{attribute 'c++_compatible'}
FUNCTION_BLOCK FB_ReadJSON IMPLEMENTS ITcJsonSaxHandler
VAR_INPUT
    myArrayInput1 : REFERENCE TO ARRAY[1..CONSt.STATION_NUMBER] OF DINT;
    myArrayInput2 : REFERENCE TO ARRAY[1..CONSt.STATION_NUMBER] OF DINT;
END_VAR
VAR_OUTPUT
END_VAR
VAR
    iArrayIndex : INT;
	iArrayNumber : INT := 0;
END_VAR

{attribute 'TcTypeSystem'}
{attribute 'no-analysis'}
{attribute 'c++_compatible'}
{attribute 'minimal_input_size' := '4'}
{attribute 'pack_mode' := '4'}
METHOD OnBool : HRESULT
VAR_INPUT
	value	: BOOL;
END_VAR
END_METHOD

{attribute 'TcTypeSystem'}
{attribute 'no-analysis'}
{attribute 'c++_compatible'}
{attribute 'minimal_input_size' := '4'}
{attribute 'pack_mode' := '4'}
METHOD OnDint : HRESULT
VAR_INPUT
	value	: DINT;
END_VAR
END_METHOD

{attribute 'TcTypeSystem'}
{attribute 'no-analysis'}
{attribute 'c++_compatible'}
{attribute 'minimal_input_size' := '4'}
{attribute 'pack_mode' := '4'}
METHOD OnEndArray : HRESULT
VAR_INPUT
	elementCount	: UDINT;
END_VAR
OnEndArray := S_OK;
END_METHOD

{attribute 'TcTypeSystem'}
{attribute 'no-analysis'}
{attribute 'c++_compatible'}
{attribute 'minimal_input_size' := '4'}
{attribute 'pack_mode' := '4'}
METHOD OnEndObject : HRESULT
VAR_INPUT
	memberCount	: UDINT;
END_VAR
OnEndObject := S_OK;
END_METHOD

{attribute 'TcTypeSystem'}
{attribute 'no-analysis'}
{attribute 'c++_compatible'}
{attribute 'minimal_input_size' := '4'}
{attribute 'pack_mode' := '4'}
METHOD OnKey : HRESULT
VAR_IN_OUT CONSTANT
	key	: STRING;
END_VAR
VAR_INPUT
	len	: UDINT;
END_VAR
OnKey := S_OK;
END_METHOD

{attribute 'TcTypeSystem'}
{attribute 'no-analysis'}
{attribute 'c++_compatible'}
{attribute 'minimal_input_size' := '4'}
{attribute 'pack_mode' := '4'}
METHOD OnLint : HRESULT
VAR_INPUT
	value	: LINT;
END_VAR
END_METHOD

{attribute 'TcTypeSystem'}
{attribute 'no-analysis'}
{attribute 'c++_compatible'}
{attribute 'minimal_input_size' := '4'}
{attribute 'pack_mode' := '4'}
METHOD OnLreal : HRESULT
VAR_INPUT
	value	: LREAL;
END_VAR
END_METHOD

{attribute 'TcTypeSystem'}
{attribute 'no-analysis'}
{attribute 'c++_compatible'}
{attribute 'minimal_input_size' := '4'}
{attribute 'pack_mode' := '4'}
METHOD OnNull : HRESULT
END_METHOD

{attribute 'TcTypeSystem'}
{attribute 'no-analysis'}
{attribute 'c++_compatible'}
{attribute 'minimal_input_size' := '4'}
{attribute 'pack_mode' := '4'}
METHOD OnRawNumber : HRESULT
VAR_IN_OUT CONSTANT
	value	: STRING;
END_VAR
VAR_INPUT
	len	: UDINT;
END_VAR
END_METHOD

{attribute 'TcTypeSystem'}
{attribute 'no-analysis'}
{attribute 'c++_compatible'}
{attribute 'minimal_input_size' := '4'}
{attribute 'pack_mode' := '4'}
METHOD OnStartArray : HRESULT
THIS^.iArrayIndex := 1;
THIS^.iArrayNumber := THIS^.iArrayNumber + 1;
OnStartArray := S_OK;
END_METHOD

{attribute 'TcTypeSystem'}
{attribute 'no-analysis'}
{attribute 'c++_compatible'}
{attribute 'minimal_input_size' := '4'}
{attribute 'pack_mode' := '4'}
METHOD OnStartObject : HRESULT
OnStartObject := S_OK;
END_METHOD

{attribute 'TcTypeSystem'}
{attribute 'no-analysis'}
{attribute 'c++_compatible'}
{attribute 'minimal_input_size' := '4'}
{attribute 'pack_mode' := '4'}
METHOD OnString : HRESULT
VAR_IN_OUT CONSTANT
	value	: STRING;
END_VAR
VAR_INPUT
	len	: UDINT;
END_VAR
END_METHOD

{attribute 'TcTypeSystem'}
{attribute 'no-analysis'}
{attribute 'c++_compatible'}
{attribute 'minimal_input_size' := '4'}
{attribute 'pack_mode' := '4'}
METHOD OnUdint : HRESULT
VAR_INPUT
	value	: UDINT;
END_VAR
IF THIS^.iArrayNumber = 1 THEN
    THIS^.myArrayInput1[THIS^.iArrayIndex] := TO_DINT(value);
    THIS^.iArrayIndex                      := THIS^.iArrayIndex + 1;
ELSIF THIS^.iArrayNumber = 2 THEN
    THIS^.myArrayInput2[THIS^.iArrayIndex] := TO_DINT(value);
    THIS^.iArrayIndex                      := THIS^.iArrayIndex + 1;
END_IF
OnUdint := S_OK;
END_METHOD

{attribute 'TcTypeSystem'}
{attribute 'no-analysis'}
{attribute 'c++_compatible'}
{attribute 'minimal_input_size' := '4'}
{attribute 'pack_mode' := '4'}
METHOD OnUlint : HRESULT
VAR_INPUT
	value	: ULINT;
END_VAR
END_METHOD

{attribute 'TcTypeSystem'}
{attribute 'no-analysis'}
{attribute 'c++_compatible'}
{attribute 'minimal_input_size' := '4'}
{attribute 'pack_mode' := '4'}
METHOD TcAddRef : UDINT
END_METHOD

{attribute 'TcTypeSystem'}
{attribute 'no-analysis'}
{attribute 'c++_compatible'}
{attribute 'minimal_input_size' := '4'}
{attribute 'pack_mode' := '4'}
METHOD TcQueryInterface : HRESULT
VAR_INPUT
	iid	: REFERENCE TO IID;
	pipItf	: POINTER TO PVOID;
END_VAR
END_METHOD

{attribute 'TcTypeSystem'}
{attribute 'no-analysis'}
{attribute 'c++_compatible'}
{attribute 'minimal_input_size' := '4'}
{attribute 'pack_mode' := '4'}
METHOD TcRelease : UDINT
END_METHOD

END_FUNCTION_BLOCK

(* stored: Version 1.1.0.1, ProductVersion 3.1.4024.6
   POU FB_ReadJSON: Id {2c20b591-6e1e-47a9-9cd2-1b0bc13d2a9c}, SpecialFunc None
   Method OnBool: Id {9a4d5a14-73d8-44e6-925f-276a9b7a4d99}
   Method OnDint: Id {b50830c8-627a-42de-8983-471ff1c6c0a0}
   Method OnEndArray: Id {f64908a6-37c0-4edc-b132-7a23c8c64f09}
   Method OnEndObject: Id {3852d89c-fafd-4e01-bb18-7e78a637b1f3}
   Method OnKey: Id {ceb41c6f-bffd-4d12-bea7-c139a1d358a7}
   Method OnLint: Id {265a7821-0589-4d69-be9b-1f75863bafc1}
   Method OnLreal: Id {a38012a6-8871-46f1-88df-17f437ec3332}
   Method OnNull: Id {2fe6e22a-8431-4936-b402-09d666003baf}
   Method OnRawNumber: Id {d9e128aa-0db5-4660-b480-33da9c1c4a78}
   Method OnStartArray: Id {6c0f6252-223d-47ac-9480-6434f3021583}
   Method OnStartObject: Id {154319f1-7500-4601-a5ac-3b43c0d5ae1f}
   Method OnString: Id {0b5aa270-bf48-441d-8d33-34dbae61aa92}
   Method OnUdint: Id {c3184c14-0ac5-463f-88be-67260d5beb5f}
   Method OnUlint: Id {d82d5f58-11ea-4618-a7f0-e07444bf9b7e}
   Method TcAddRef: Id {18707b48-7fec-4fa6-9f12-d207fcb3eb6f}
   Method TcQueryInterface: Id {16562a11-f047-4804-80e4-ce6a68573a0b}
   Method TcRelease: Id {b6583a91-d3cd-4b37-989f-1b67963bf2ea} *)
